{attribute 'qualified_only'}
{attribute 'strict'}
TYPE E_TIME_MODE :
(
	LOCAL	:= 0,
	UTC		:= 1
);
END_TYPE

(* stored: Version 1.1.0.1, ProductVersion 3.1.4022.16
   DUT E_TIME_MODE: Id {8d99a6b2-d9af-4a3c-b6db-25205bf8f61d} *)
